{attribute 'GeneratedUsingTerminal: EL4002-0000-0016'}
{attribute addProperty BoxType "EL4002-0000-0016"}
{attribute addProperty Id "AO_Outputs_Channel_1AT %Q*AO_Output_Channel_BA7EBB7C2AO_Outputs_Channel_2AT %Q*AO_Output_Channel_BA7EBB7C2WcStateAT %I*WcState_0B2B16F91InfoDataAT %I*InfoData_94A18F5E2"}
{attribute addProperty CRC "3400845557"}
{attribute addProperty Size "7"}
TYPE EL4002_CAB4C8F5 EXTENDS EtcSlaveTerminalBase_947E5A46 :
STRUCT
	{attribute addProperty Name "AO_Outputs_Channel_1"}
	AO_Outputs_Channel_1 : AO_Output_Channel_BA7EBB7C;
	{attribute addProperty Name "AO_Outputs_Channel_2"}
	AO_Outputs_Channel_2 : AO_Output_Channel_BA7EBB7C;
	{attribute addProperty Name "WcState"}
	WcState : WcState_0B2B16F9;
	{attribute addProperty Name "InfoData"}
	InfoData : InfoData_94A18F5E;
END_STRUCT
END_TYPE

(* stored: Version 1.2.0.0, ProductVersion 3.1.4024.9
   DUT EL4002_CAB4C8F5: Id {65707458-daf0-47ae-984a-b78ee7b5ba56} *)
